RoboDK station: Rollercoaster Sim Robbie Vandeputte.rdk

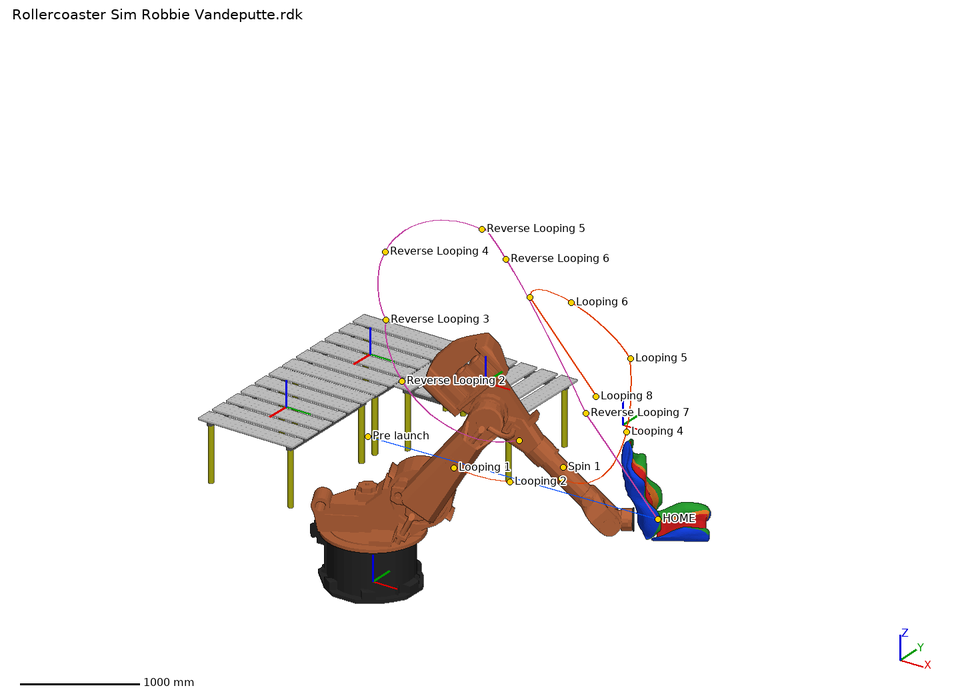
[picture v0: the station drawn from its stored meshes, robots at their saved joint values, targets as dots, program paths as lines]
Station Rollercoaster Sim Robbie Vandeputte (saved by RoboDK 5.9.5). Poses are relative to the parent item; angles as X-Y-Z fixed-axis rotations.
  - frame KUKA KR 150 L120/2 Base at (0, 0, 0) mm
    - robot KUKA KR 150 L120/2: 6 axes, payload 120 kg, reach 2810 mm, repeatability 0.2 mm, weight 1140 kg
        modified DH rows (alpha deg, a mm, theta deg, d mm): 0, 0, 0, 865; -90, 410, 0, 0; 0, 1000, -90, 0; -90, 45, 0, 1400; 90, 0, 0, 0; -90, 0, 180, 210
        joint limits [-185, -130, -120, -350, -120, -350] to [185, 3, 148, 350, 120, 350]; home [0, -90, 90, 0, 0, 0]; saved at [-27.738, -54.678, 100.891, -171.556, 46.525, 174.168]
      - tool recaro, TCP at (0, 0, 200) mm, size 836.7 x 528.2 x 740.8 mm, geometry from recaro.IGS
  - frame Frame 2 at (-1800, 1305.45, 600) mm, rotated rx 0 ry 0 rz -90 deg
    - object Object Table at (0, 0, 0) mm, size 1193.8 x 965.2 x 609.6 mm, geometry from Object Table.wrl
    - target HOME (Cartesian target) at (151.11, 3901.3, 101.37) mm, rotated rx 0 ry 90 rz 123.85 deg; joints [-27.738, -54.678, 100.891, -171.556, 46.525, 174.168] of KUKA KR 150 L120/2
    - target Pre launch (Cartesian target) at (147.79, 938.19, 42.43) mm, rotated rx 116.28 ry 84.26 rz -111.96 deg; joints [-142.843, -73.93, 132.07, -280.672, 93.595, 206.127] of KUKA KR 150 L120/2
    - target Looping 1 (Cartesian target) at (-33.09, 1690.15, -110) mm, rotated rx 3.07 ry 88.9 rz 103.8 deg; joints [-112.103, -65.543, 134.784, -280.262, 95.039, 200.357] of KUKA KR 150 L120/2
    - target Looping 2 (Cartesian target) at (-82.59, 2226.59, -109.33) mm, rotated rx -58.82 ry 54.26 rz 27.26 deg; joints [-88.513, -56.81, 131.049, -262.606, 106.217, 228.032] of KUKA KR 150 L120/2
    - target Looping 3 (Cartesian target) at (-35.21, 2784.4, 97.2) mm, rotated rx -36.73 ry 55.55 rz 25.24 deg; joints [-66.402, -59.423, 121.391, -255.737, 113.14, 233.035] of KUKA KR 150 L120/2
    - target Looping 4 (Cartesian target) at (612.16, 3903.08, 1099.01) mm, rotated rx -16.55 ry 36.56 rz 35.24 deg; joints [-23.574, -72.442, 92.379, -210.301, 83.785, 249.025] of KUKA KR 150 L120/2
    - target Looping 5 (Cartesian target) at (756.65, 4044.4, 1878.6) mm, rotated rx -6.38 ry -14.59 rz 13.63 deg; joints [-11.147, -59.873, 47.059, -164.437, 71.88, 264.157] of KUKA KR 150 L120/2
    - target Looping 6 (Cartesian target) at (995.04, 3609.13, 2375.82) mm, rotated rx -8.88 ry -45.82 rz 18.41 deg; joints [-0.461, -69.453, 31.733, -129.195, 68.609, 229.184] of KUKA KR 150 L120/2
    - target Looping 7 (Cartesian target) at (737.49, 3004.37, 2154.41) mm, rotated rx 145.66 ry -46.48 rz -120.4 deg; joints [-10.649, -85.518, 33.885, -70.53, 119.747, 253.528] of KUKA KR 150 L120/2
    - target Looping 8 (Cartesian target) at (-151.77, 3058.7, 890.05) mm, rotated rx 157.1 ry -3.52 rz -145.27 deg; joints [-49.744, -92.6, 94.316, 2.914, 65.298, 253.596] of KUKA KR 150 L120/2
    - target Spin 1 (Cartesian target) at (-27.43, 2809.52, 213.93) mm, rotated rx 180 ry -3.52 rz -145 deg; joints [-52.035, -89.458, 118.57, -3.889, 59.914, 254.886] of KUKA KR 150 L120/2
    - target Spin 2 (Cartesian target) at (-27.43, 2809.52, 213.94) mm, rotated rx -176.6 ry 0.89 rz 110.28 deg; joints [-52.035, -89.458, 118.57, -3.889, 59.914, -209.855] of KUKA KR 150 L120/2
    - target Spin 3 (Cartesian target) at (-27.43, 2809.52, 213.94) mm, rotated rx 178.87 ry 3.33 rz 16.23 deg; joints [-52.035, -89.458, 118.57, -3.889, 59.914, -303.847] of KUKA KR 150 L120/2
    - target Spin 4 (Cartesian target) at (-27.43, 2809.52, 213.94) mm, rotated rx 176.66 ry -1.1 rz -73.22 deg; joints [-52.035, -89.458, 118.57, -183.889, -59.914, -213.362] of KUKA KR 150 L120/2
    - target Spin 5 (Cartesian target) at (-27.43, 2809.52, 213.94) mm, rotated rx 178.72 ry -3.28 rz -123.69 deg; joints [-52.035, -89.458, 118.57, -183.889, -59.914, -263.84] of KUKA KR 150 L120/2
    - target Reverse Looping 1 (Cartesian target) at (-183.06, 2254.59, 241.35) mm, rotated rx 176.85 ry -1.57 rz -81.38 deg; joints [-72.28, -97.585, 125.046, -183.219, -60.445, -242.166] of KUKA KR 150 L120/2
    - target Reverse Looping 2 (Cartesian target) at (-4.08, 1182.8, 567.46) mm, rotated rx 174.07 ry -57.87 rz -76.44 deg; joints [-101.379, -111.933, 130.72, -240.529, -76.246, -252.51] of KUKA KR 150 L120/2
    - target Reverse Looping 3 (Cartesian target) at (46.25, 1051.75, 1118.22) mm, rotated rx 11.65 ry -74.21 rz 87.31 deg; joints [-105.149, -115.483, 123.833, -286.153, -86.75, -257.139] of KUKA KR 150 L120/2
    - target Reverse Looping 4 (Cartesian target) at (79.9, 1070.09, 1772.21) mm, rotated rx 3.19 ry -9.24 rz 98.02 deg; joints [62.019, -116.667, -52.888, -170.063, -79.572, -252.102] of KUKA KR 150 L120/2
    - target Reverse Looping 5 (Cartesian target) at (-32.34, 1973.53, 2191.34) mm, rotated rx 34.88 ry 65.05 rz 105.33 deg; joints [-97.017, -94.249, 61.895, -56.71, -101.654, -243.716] of KUKA KR 150 L120/2
    - target Reverse Looping 6 (Cartesian target) at (768.94, 2783.95, 2456.38) mm, rotated rx 132.98 ry 60.9 rz -172.75 deg; joints [-48.498, -79.047, 7.027, -105.153, -105.474, -220.566] of KUKA KR 150 L120/2
    - target Reverse Looping 7 (Cartesian target) at (1371.29, 4018.29, 1609.12) mm, rotated rx 152.26 ry 40.15 rz -148.33 deg; joints [-0.982, -73.129, 46.651, -164.512, -71.491, -227.825] of KUKA KR 150 L120/2
  - frame Frame 3 at (-700, 2645.45, 600) mm
    - object Object Table at (0, 0, 0) mm, size 1193.8 x 965.2 x 609.6 mm, geometry from Object Table.wrl
  - frame Frame 4 at (-1800, 2531.01, 600) mm, rotated rx 0 ry 0 rz -90 deg
    - object Object Table at (0, 0, 0) mm, size 1193.8 x 965.2 x 609.6 mm, geometry from Object Table.wrl
  - program Prelaunch (4 instructions, listed below)
  - program Looping (7 instructions, listed below)
  - program Spin (7 instructions, listed below)
  - program Reverse looping (7 instructions, listed below)
  - program MAIN (4 instructions, listed below)
  - frame Frame 5 at (0, 3645.45, 0) mm
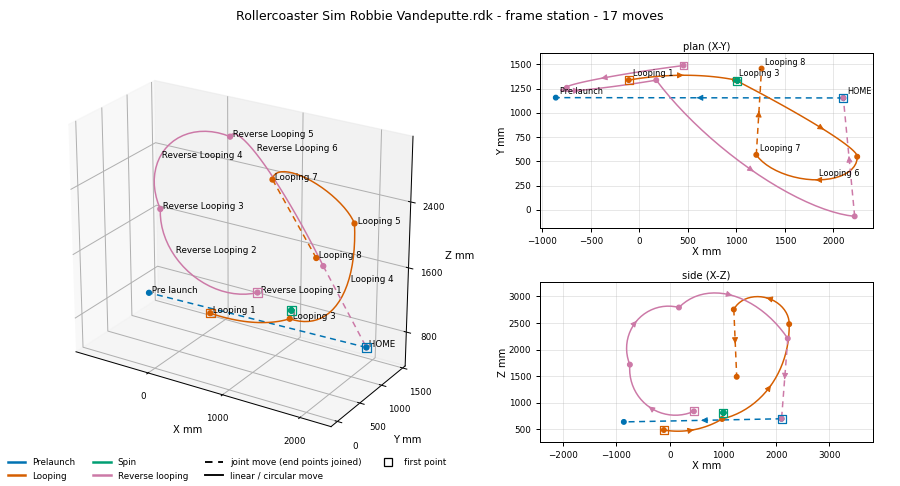
[picture p0: tool path of Rollercoaster Sim Robbie Vandeputte.rdk in frame station, 17 of 17 moves have a stored position in this frame; points joined in program order, loops and branches not executed]

--- program Prelaunch (robot KUKA KR 150 L120/2) ---
  Set Ref.: Frame 2
  Set Tool: recaro
  MoveJ (HOME)
  MoveJ (Pre launch)

--- program Looping (robot KUKA KR 150 L120/2) ---
  Set Ref.: Frame 2
  Set Tool: recaro
  MoveJ (Looping 1)
  MoveC (Looping 2, Looping 3)
  MoveC (Looping 4, Looping 5)
  MoveC (Looping 6, Looping 7)
  MoveJ (Looping 8)

--- program Spin (robot KUKA KR 150 L120/2) ---
  Set Ref.: Frame 2
  Set Tool: recaro
  MoveJ (Spin 1)
  MoveL (Spin 2)
  MoveL (Spin 3)
  MoveL (Spin 4)
  MoveL (Spin 5)

--- program Reverse looping (robot KUKA KR 150 L120/2) ---
  Set Ref.: Frame 2
  Set Tool: recaro
  MoveL (Reverse Looping 1)
  *MoveC (Reverse Looping 2, Reverse Looping 3)
  *MoveC (Reverse Looping 4, Reverse Looping 5)
  *MoveC (Reverse Looping 6, Reverse Looping 7)
  MoveJ (HOME)

--- program MAIN (robot KUKA KR 150 L120/2) ---
  Call Prelaunch
  Call Looping
  Call Spin
  Call Reverse looping
